// TIA Portal project "S120 Motion Control" (V15.1)

(* hardware
DEVICE "S71500/ET200MP station_1"  S7-1500 station
   slot 0: "Rail_0"  Rack  6ES7 590-1***0-0AA0
   slot 1: "PLC_1"  CPU 1512C-1 PN  6ES7 512-1CK01-0AB0  V2.6
      slot 3: "CPU display_1"  6ES7591-1AA00-0AA0
DEVICE "GSD device_1"  GSD.Device.PN
   slot 0: "Rack"  Rack  V1.0
   slot 0: "SINAMICS-S120-CU310-2PN"  SINAMICS S120 CU310-2 PN V4.8  6SL3 040-1LA01-0AAx  V4.80
      slot 0: "SINAMICS S120 CU310-2 PN V4.8"  SINAMICS S120 CU310-2 PN V4.8
      slot 1: "PN-IO"  PN-IO
         slot 1: "Port 1"  Port 1
         slot 2: "Port 2"  Port 2
   slot 1: "DO SERVO_1"  DO SERVO
      slot 0: "Module Access Point"  Module Access Point
   slot 2: "SIEMENS telegram 105, PZD-10/10"  SIEMENS telegram 105, PZD-10/10
*)

// ===== PLC "PLC_1"  CPU 1512C-1 PN =====

VAR_GLOBAL   // PLC tag table "Default tag table"
   "System_Byte" AT %MB1 : Byte;
   "FirstScan" AT %M1.0 : Bool;
   "DiagStatusUpdate" AT %M1.1 : Bool;
   "AlwaysTRUE" AT %M1.2 : Bool;
   "AlwaysFALSE" AT %M1.3 : Bool;
   "Clock_Byte" AT %MB0 : Byte;
   "Clock_10Hz" AT %M0.0 : Bool;
   "Clock_5Hz" AT %M0.1 : Bool;
   "Clock_2.5Hz" AT %M0.2 : Bool;
   "Clock_2Hz" AT %M0.3 : Bool;
   "Clock_1.25Hz" AT %M0.4 : Bool;
   "Clock_1Hz" AT %M0.5 : Bool;
   "Clock_0.625Hz" AT %M0.6 : Bool;
   "Clock_0.5Hz" AT %M0.7 : Bool;
   "System_Byte(1)" AT %MB1 : Byte;
   "MotionControl_Poition_Actor_Interface_AddressIn" AT %I126.0 : "PD_TEL105_IN";
   "MotionControl_Poition_Actor_Interface_AddressOut" AT %Q128.0 : "PD_TEL105_OUT";
   "Power" AT %M2.0 : Bool;
   "execute" AT %M2.1 : Bool;
   "done1" AT %M2.2 : Bool;
   "done2" AT %M2.3 : Bool;
   "execute2" AT %M2.4 : Bool;
   "Timer1" AT %MD4 : Time;
   "done3" AT %M2.5 : Bool;
   "done4" AT %M2.6 : Bool;
   "Timer2" AT %MD8 : Time;
   "execute3" AT %M2.7 : Bool;
   "done5" AT %M3.0 : Bool;
   "Start Power" AT %M3.1 : Bool;
   "Start execute" AT %M3.2 : Bool;
END_VAR

DATA_BLOCK "MC_Code_DB"   // DB3
{ S7_Optimized_Access := 'TRUE' }
VERSION : 0.1
// stored: InstanceOfName MC_Code
"MC_Code"
BEGIN
END_DATA_BLOCK

DATA_BLOCK "MC_Block_DB"   // DB4
{ S7_Optimized_Access := 'TRUE' }
VERSION : 0.1
// stored: InstanceOfName MC_Block
"MC_Block"
BEGIN
END_DATA_BLOCK

DATA_BLOCK "MotionControl_Poition"   // DB1, Motion_DB
{ S7_Optimized_Access := 'TRUE' }
AUTHOR : SIMATIC
FAMILY : MC_1500
VERSION : 4.0
// stored: InstanceOfName TO_PositioningAxis
"TO_PositioningAxis"
BEGIN
END_DATA_BLOCK

FUNCTION_BLOCK "MC_Block"   // FB1, LAD
{ S7_Optimized_Access := 'TRUE' }
VERSION : 0.1
   VAR
      MC_POWER_Instance : MC_POWER;
      IEC_Timer_0_Instance : TON_TIME;
      MC_MOVERELATIVE_Instance : MC_MOVERELATIVE;
      MC_MOVERELATIVE_Instance_1 : MC_MOVERELATIVE;
      MC_MOVERELATIVE_Instance_2 : MC_MOVERELATIVE;
      MC_MOVERELATIVE_Instance_3 : MC_MOVERELATIVE;
      MC_HALT_Instance : MC_HALT;
      IEC_Timer_0_Instance_1 : TON_TIME;
      MC_HALT_Instance_1 : MC_HALT;
      IEC_Timer_0_Instance_2 : TON_TIME;
      MC_MOVERELATIVE_Instance_4 : MC_MOVERELATIVE;
   END_VAR
BEGIN

REGION Network 1
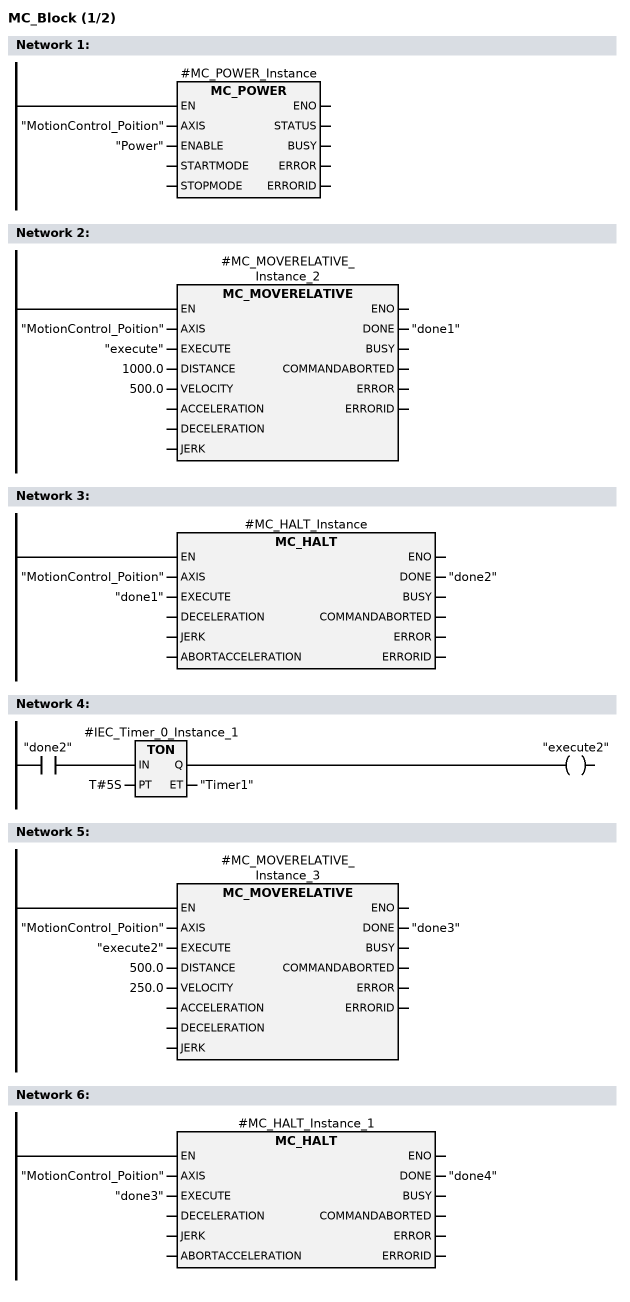
   #MC_POWER_Instance(Axis := "MotionControl_Poition", Enable := "Power");   // MC_POWER
END_REGION

REGION Network 2
   #MC_MOVERELATIVE_Instance_2(Axis := "MotionControl_Poition",   // MC_MOVERELATIVE
                           Execute := "execute",
                           Distance := 1000.0,
                           Velocity := 500.0,
                           Done => "done1");
END_REGION

REGION Network 3
   #MC_HALT_Instance(Axis := "MotionControl_Poition", Execute := "done1", Done => "done2");   // MC_HALT
END_REGION

REGION Network 4
   #IEC_Timer_0_Instance_1(IN := "done2", PT := T#5S, ET => "Timer1");   // TON
   "execute2" := #IEC_Timer_0_Instance_1.Q;
END_REGION

REGION Network 5
   #MC_MOVERELATIVE_Instance_3(Axis := "MotionControl_Poition",   // MC_MOVERELATIVE
                           Execute := "execute2",
                           Distance := 500.0,
                           Velocity := 250.0,
                           Done => "done3");
END_REGION

REGION Network 6
   #MC_HALT_Instance_1(Axis := "MotionControl_Poition", Execute := "done3", Done => "done4");   // MC_HALT
END_REGION

REGION Network 7
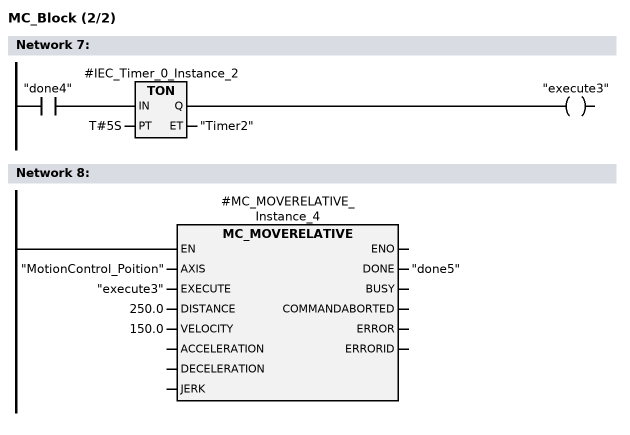
   #IEC_Timer_0_Instance_2(IN := "done4", PT := T#5S, ET => "Timer2");   // TON
   "execute3" := #IEC_Timer_0_Instance_2.Q;
END_REGION

REGION Network 8
   #MC_MOVERELATIVE_Instance_4(Axis := "MotionControl_Poition",   // MC_MOVERELATIVE
                           Execute := "execute3",
                           Distance := 250.0,
                           Velocity := 150.0,
                           Done => "done5");
END_REGION
END_FUNCTION_BLOCK

FUNCTION_BLOCK "MC_Code"   // FB2, LAD
{ S7_Optimized_Access := 'TRUE' }
VERSION : 0.1
BEGIN

REGION Network 1
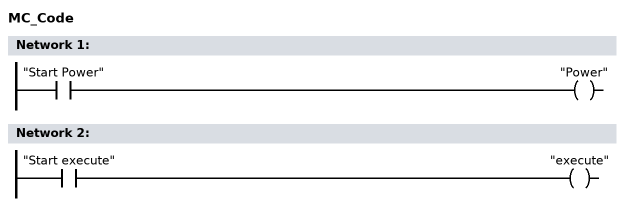
   RUNG wire#powerrail
      Contact( "Start Power" )
      Coil( "Power" )
   END_RUNG
   // the same network as SCL:
   "Power" := "Start Power";
END_REGION

REGION Network 2
   RUNG wire#powerrail
      Contact( "Start execute" )
      Coil( "execute" )
   END_RUNG
   // the same network as SCL:
   "execute" := "Start execute";
END_REGION
END_FUNCTION_BLOCK

ORGANIZATION_BLOCK "Main"   // OB1, LAD, ProgramCycle
TITLE = "Main Program Sweep (Cycle)"
{ S7_Optimized_Access := 'TRUE' }
VERSION : 0.1
   VAR_INPUT
      Initial_Call : Bool;   // Initial call of this OB
      Remanence : Bool;   // =True, if remanent data are available
   END_VAR
BEGIN

REGION Network 1
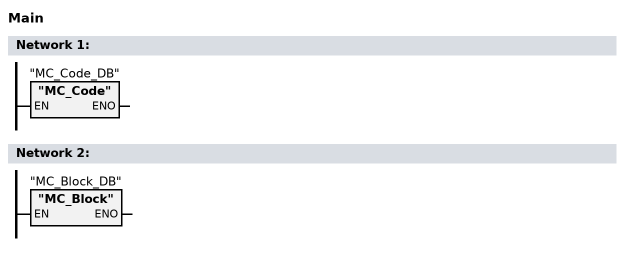
   RUNG wire#powerrail
      "MC_Code_DB"()
   END_RUNG
   // the same network as SCL:
   "MC_Code_DB"();   // "MC_Code"
END_REGION

REGION Network 2
   RUNG wire#powerrail
      "MC_Block_DB"()
   END_RUNG
   // the same network as SCL:
   "MC_Block_DB"();   // "MC_Block"
END_REGION
END_ORGANIZATION_BLOCK